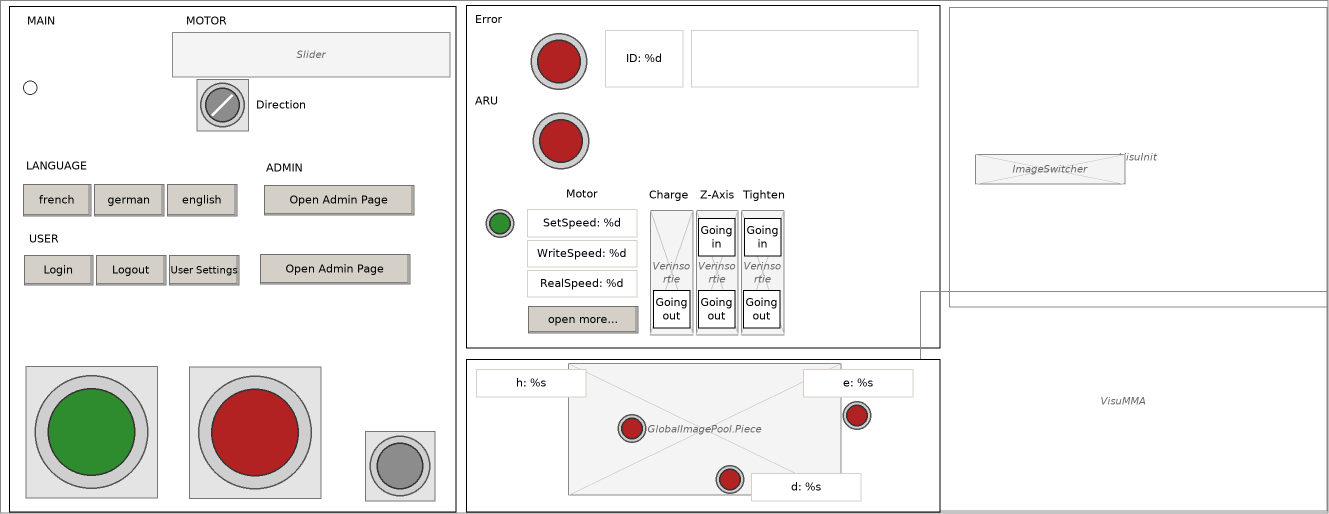
VISUALIZATION Visualization  // 1329x514
    Rectangle (466,5 474x343)
    Rectangle (9,6 447x506)
    Label (24,6 80x30), "MAIN"
    Lamp1 (527,108 68x66), variable: fbBtn.xAru=0, style: Lamp-Lamp1-Red
    Label (472,87 87x28), "ARU"
    RadioButton (21,39 150x97), variable: stParam.stStatus.eMMA
        Areas[0]: Text=Mode Init
        Areas[1]: Text=Mode Auto
        Areas[2]: Text=Mode Manual
    Frame (949,7 378x300), frame switch variable: stParam.stStatus.eMMA
        shows VisuInit()
        shows VisuAuto()
        shows VisuManual()
        shows VisuMMA()
    Frame (920,291 407x220)
        shows VisuMMA()
    Lamp1 (526,27 66x69), variable: stParam.stStatus.xErreur, style: Lamp-Lamp1-Red
    Label (472,5 55x29), "Error"
    Textfield (691,30 227x57), text variable: stParam.stStatus.sMessage, text list: 'ErrorList', text index: stParam.stStatus.iId
    Textfield (605,30 78x57), "ID: %d", text variable: stParam.stStatus.iId
    PushSwitch (24,366 135x132), tooltip "Start", variable: stIO.stIn.xStartIO, behaviour: TAP, style: Switch-PushSwitch-Green
    PushSwitch (189,364 132x137), tooltip "Stop", variable: stIO.stIn.xStopIO, invisible if: fbMMA.iEtape<>350, behaviour: TAP, style: Switch-PushSwitch-Red
    PushSwitch (365,431 70x70), tooltip "Reset", variable: stIO.stIn.xResetIO, behaviour: TAP, style: Switch-PushSwitch-Gray
    Slider (172,32 278x45), variable: stIO.stIn.lSetSpeedMotor, scale 100..1500
    Label (183,6 80x30), "MOTOR"
    Label (253,90 117x30), "Direction"
    RotarySwitch (195,79 55x52), variable: stIO.stIn.xMotorDirection, behaviour: TOGGLE, style: Switch-RotarySwitch-Gray
    Button (264,185 150x30), "Open Admin Page"
        OnMouseClick: change screen: VisuAdmin
    Label (263,153 80x30), "ADMIN"
    Button (23,184 68x32), "french"
        OnMouseClick: ChangeLanguage ChangeLanguage=fr
    Label (23,151 80x30), "LANGUAGE"
    Button (94,184 70x32), "german"
        OnMouseClick: ChangeLanguage ChangeLanguage=de
    Button (167,184 70x32), "english"
        OnMouseClick: ChangeLanguage ChangeLanguage=en
    Label (724,180 80x30), "Tighten"
    Label (629,180 80x30), "Charge"
    Label (677,180 80x30), "Z-Axis"
    Image (741,210 43x125), invisible if: fbAct3.xInInPos=0, image: Verinrentree
    Image (696,210 42x125), invisible if: fbAct2.xInInPos=0, image: Verinrentree
    Image (650,210 43x125), invisible if: fbAct1.xInInPos=0, image: Verinrentree
    Image (650,210 43x125), invisible if: fbAct1.xInOutPos=0, image: Verinsortie
    Image (696,210 42x125), invisible if: fbAct2.xInOutPos=0, image: Verinsortie
    Image (741,210 43x125), invisible if: fbAct3.xInOutPos=0, image: Verinsortie
    Rectangle (743,290 37x38), "Going out", invisible if: fbAct3.xGoingOutNow=0
    Rectangle (698,290 37x38), "Going out", invisible if: fbAct2.xGoingOutNow=0
    Rectangle (653,290 37x38), "Going out", invisible if: fbAct1.xGoingOutNow=0
    Rectangle (744,218 37x38), "Going in", invisible if: fbAct3.xGoingInNow=0
    Rectangle (698,218 37x38), "Going in", invisible if: fbAct2.xGoingInNow=0
    Label (527,179 110x30), "Motor"
    Lamp1 (482,207 36x33), variable: fbMotor.xOnOff, style: Lamp-Lamp1-Green
    Textfield (527,209 110x28), "SetSpeed: %d", text variable: fbMotor.Consigne
    Textfield (527,270 110x27), "RealSpeed: %d", text variable: fbMotor.fbConvertTachoToNumSpeed.lrValeur
    Button (528,306 110x27), "open more..."
        OnMouseClick: change screen: VisuMotor
    Textfield (527,240 110x27), "WriteSpeed: %d", text variable: fbMotor.fbConvertNumToMotorOut.lrConsigne
    Rectangle (466,359 474x153)
    Image (568,363 273x132), image: GlobalImagePool.Piece
    Textfield (803,369 110x28), "e: %s", text variable: fbTCP.OutputGlobal.Resulte
        p3092690914: fbTCP.OutputGlobal.Boole
    Textfield (476,369 110x28), "h: %s", text variable: fbTCP.OutputGlobal.Resulth
    Textfield (751,473 110x28), "d: %s", text variable: fbTCP.OutputGlobal.Resultd
    Lamp1 (614,412 36x33), variable: fbTCP.OutputGlobal.Boolh=0, style: Lamp-Lamp1-Red
    Lamp1 (839,399 36x33), variable: fbTCP.OutputGlobal.Boole=0, style: Lamp-Lamp1-Red
    Lamp1 (712,463 36x33), variable: fbTCP.OutputGlobal.Boold=0, style: Lamp-Lamp1-Red
    ImageSwitcher (975,154 150x30), behaviour: TOGGLE
    Button (382,261 1x2)
    Button (24,255 69x30), "Login"
        OnMouseClick: VisuUserMgmt Type=Login
    Button (96,255 70x30), "Logout"
        OnMouseClick: VisuUserMgmt Type=Logout
    Label (26,224 80x30), "USER"
    Button (169,255 70x30), "User Settings"
        OnMouseClick: VisuUserMgmt Type=OpenUserConfiguration
    Button (260,254 150x30), "Open Admin Page"
        OnMouseClick: change screen: Vi_Alarmes
END_VISUALIZATION

(* stored: Version 1.1.0.1, ProductVersion 3.1.4020.6
   Visu Visualization: Id {1e4c2f99-d035-41f9-adba-3d4322eca24e} *)
